// TIA Portal V19 export
VAR_GLOBAL   // PLC tag table "Default tag table"
   B0 AT %QB0 : Byte;
   B1 AT %QB1 : Byte;
   Clock_Byte AT %MB0 : Byte;
   Clock_10Hz AT %M0.0 : Bool;
   Clock_5Hz AT %M0.1 : Bool;
   "Clock_2.5Hz" AT %M0.2 : Bool;
   Clock_2Hz AT %M0.3 : Bool;
   "Clock_1.25Hz" AT %M0.4 : Bool;
   Clock_1Hz AT %M0.5 : Bool;
   "Clock_0.625Hz" AT %M0.6 : Bool;
   "Clock_0.5Hz" AT %M0.7 : Bool;
   System_Byte AT %MB1 : Byte;
   FirstScan AT %M1.0 : Bool;
   DiagStatusUpdate AT %M1.1 : Bool;
   AlwaysTRUE AT %M1.2 : Bool;
   AlwaysFALSE AT %M1.3 : Bool;
   "from et200sp PLC_1" AT %IB100 : Byte;
   toET200spfromPLC1 AT %QB100 : Byte;
   "from et200sp PLC_1 Right" AT %IB200 : Byte;
   "toET200spfromPLC1 Right" AT %QB200 : Byte;
END_VAR
